Omron CX-Programmer project 新工程 (CX-Programmer 9.73)

# PLC 新PLC1: CPM1(CPM1A) CPU20

## Global symbols (name address type ; comment)
0.00 BOOL  ; 摇动检测
0.01 BOOL  ; 自动
0.02 BOOL  ; 泵手动
0.03 BOOL  ; 摇动手动
0.04 BOOL  ; 超声波手动
0.05 BOOL  ; 阀门手动
0.06 BOOL  ; 循环启动
0.07 BOOL  ; 超声波定时
0.08 BOOL  ; 摇动定时
0.09 BOOL  ; 非常停止
0.10 BOOL  ; 液位检测
0.11 BOOL  ; 过载保护
10.04 BOOL  ; 泵驱动
10.05 BOOL  ; 摇动马达
10.06 BOOL  ; 超声波
10.07 BOOL  ; 卸油阀
15.00 BOOL  ; 液位正常
200.00 BOOL  ; 循环启动了
200.01 BOOL  ; 循环开始指令
200.02 BOOL  ; 泵起动
200.03 BOOL  ; 阀门闭
200.04 BOOL  ; 泵、阀门、液位异常
200.05 BOOL  ; 液有了
200.06 BOOL  ; 液位异常
200.07 BOOL  ; 泵停止
200.09 BOOL  ; 超声波开
200.10 BOOL  ; 超声波关
200.11 BOOL  ; 泵起动2
200.12 BOOL  ; 摇动开
200.13 BOOL  ; 阀门开
200.14 BOOL  ; 泵停止2
201.00 BOOL  ; 喷淋循环启动
201.01 BOOL  ; 喷淋循环开始
201.02 BOOL  ; 阀门闭2
201.03 BOOL  ; 阀门开2
201.04 BOOL  ; 泵起动3
201.05 BOOL  ; 泵停止3
201.07 BOOL  ; 喷淋循环结束
201.08 BOOL  ; 停止位到
201.09 BOOL  ; 摇动异常
201.10 BOOL  ; 液位异常
210.00 BOOL  ; 全异常
5.00 BOOL  ; 转自动
5.01 BOOL  ; 转手动
5.02 BOOL  ; 泵手动开
5.03 BOOL  ; 泵手动关
5.04 BOOL  ; 摇动手动开
5.05 BOOL  ; 摇动手动关
5.06 BOOL  ; 超声波手动开
5.07 BOOL  ; 超声波手动关
5.08 BOOL  ; 阀门手动开
5.09 BOOL  ; 阀门手动关
5.10 BOOL  ; 循环启动指令
DM1000 CHANNEL  ; 摇动计数
TIM017 BOOL  ; 喷淋时间
TIM021 BOOL  ; 全停止

## Program 大摇动 (no task)
; 【项目概况】 / 代码控制超声波清洗机，通过泵驱动、摇动马达、超声波和卸油阀的协同工作，实现工件的清洁。系统支持自动模式和手动模式。 / 系统包括PLC控制器CPM1 CPU20、泵驱动、摇动马达、超声波发生器、卸油阀、液位传感器、过载保护开关和非常停止按钮等物理设备。 / 【运行解析】 / 1.操作员可以通过自动模式选择切换运行模式。 / 2.在自动模式下，按下循环启动按钮会置位清洗循环启动标志。 / 3.在启动清洗循环前，液位传感器必须检测到液位正常标志为真，确保清洗液充足，否则无法启动。 / 4.清洗开始后，泵启动标志激活泵驱动循环清洗液，同时阀门关闭标志关闭卸油阀，保持液位稳定。 / 5.随后，系统进入超声波和摇动阶段，超声波启动标志启动超声波发生器，运行时间由超声波定时开关控制；接着摇动启动标志启动摇动马达，运行时间由摇动定时开关决定。 / 6.系统通过互锁逻辑确保超声波发生器和摇动马达不会同时运行，以避免干扰或设备过载。 / 7.摇动马达运行时，摇动计数器记录频率，若未在规定时间内达到5次，摇动异常标志会置位，表示检测到异常。 / 8.超声波和摇动完成后，喷淋循环启动标志触发喷淋清洗，泵启动3标志再次启动泵驱动，阀门关闭2标志和阀门开启2标志协作控制卸油阀，喷淋时间定时器计时300个单位后，喷淋循环结束标志置位。 / 9.最终，全停止定时器计时结束，停止位到标志置位，所有动作停止。 / 10.在手动模式下，操作员可通过泵手动开关、摇动手动开关、超声波手动开关和阀门手动开关独立控制设备。 / 11.系统通过互锁逻辑确保泵驱动和卸油阀不会同时运行，以防止清洗液同时循环和排放。 / 12.当泵手动开指令和阀门手动开指令同时置位时，系统通过优先级逻辑或互锁机制确保泵驱动和卸油阀不会同时运行。 / 13.系统通过过载保护开关和非常停止按钮监控安全状态，若触发全异常标志，所有动作立即停止。 / 14.同时，清洗循环启动标志和喷淋循环启动标志会复位到初始状态，确保设备安全复位。 / 15.液位异常标志、泵阀液位异常标志或摇动异常标志也能触发全异常标志，提供多重保护。

### Section 段1

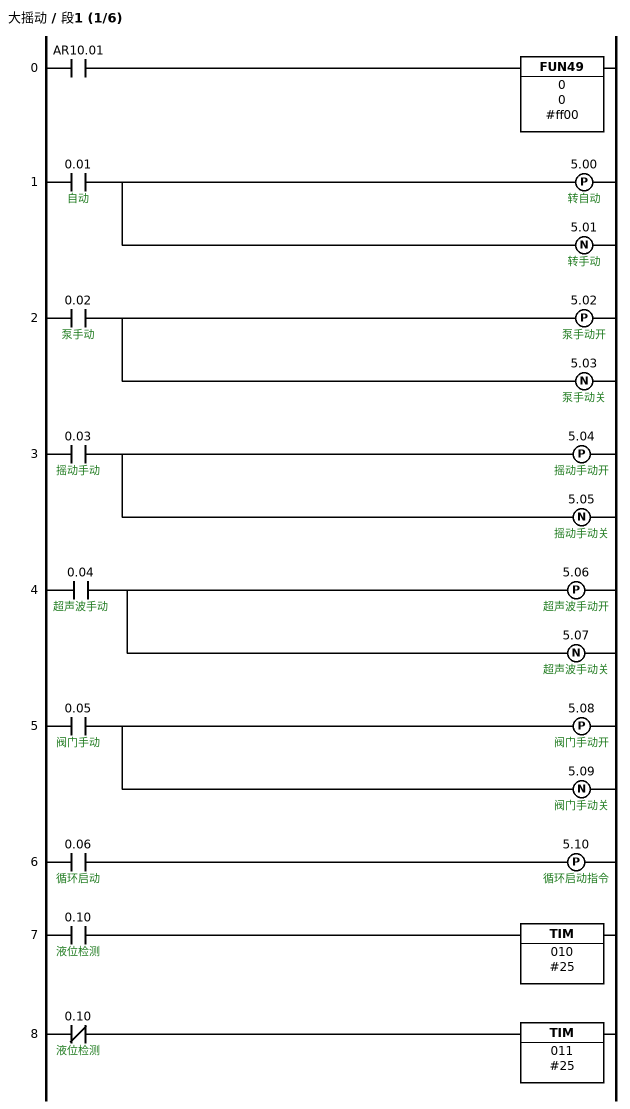
; rung 0
LD AR10.01
FUN49 0 0 #ff00
; rung 1
LD 0.01  ; 自动
DIFU(13) 5.00  ; 转自动
DIFD(14) 5.01  ; 转手动
; rung 2
LD 0.02  ; 泵手动
DIFU(13) 5.02  ; 泵手动开
DIFD(14) 5.03  ; 泵手动关
; rung 3
LD 0.03  ; 摇动手动
DIFU(13) 5.04  ; 摇动手动开
DIFD(14) 5.05  ; 摇动手动关
; rung 4
LD 0.04  ; 超声波手动
DIFU(13) 5.06  ; 超声波手动开
DIFD(14) 5.07  ; 超声波手动关
; rung 5
LD 0.05  ; 阀门手动
DIFU(13) 5.08  ; 阀门手动开
DIFD(14) 5.09  ; 阀门手动关
; rung 6
LD 0.06  ; 循环启动
DIFU(13) 5.10  ; 循环启动指令
; rung 7
LD 0.10  ; 液位检测
TIM 010 #25
; rung 8
LDNOT 0.10  ; 液位检测
TIM 011 #25

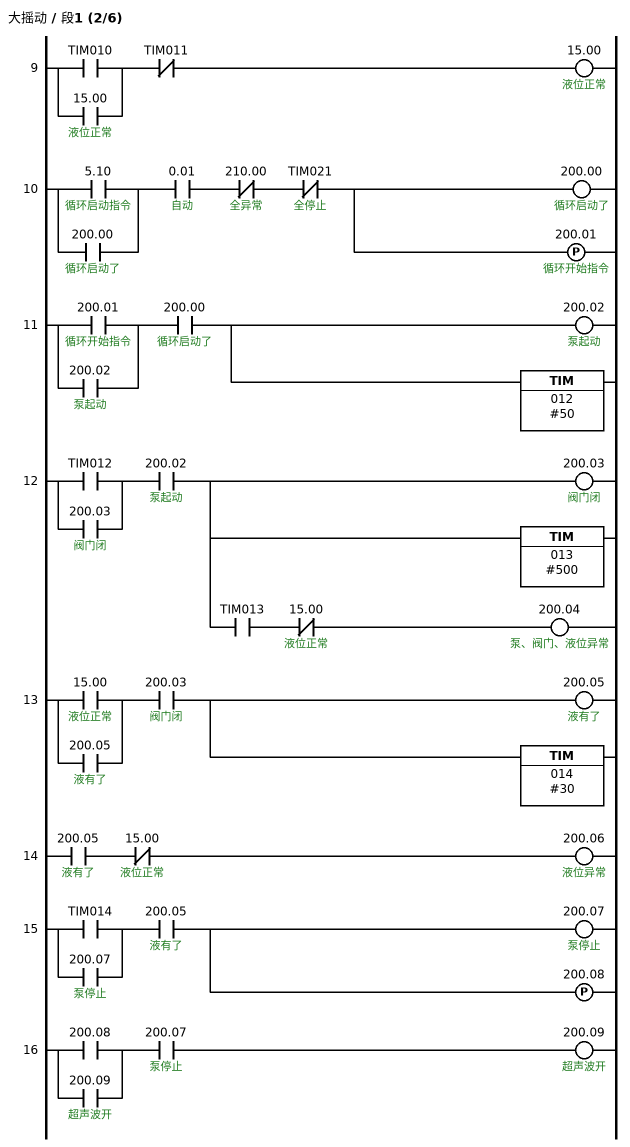
; rung 9
LD TIM010
OR 15.00  ; 液位正常
ANDNOT TIM011
OUT 15.00  ; 液位正常
; rung 10
LD 5.10  ; 循环启动指令
OR 200.00  ; 循环启动了
AND 0.01  ; 自动
ANDNOT 210.00  ; 全异常
ANDNOT TIM021  ; 全停止
OUT 200.00  ; 循环启动了
DIFU(13) 200.01  ; 循环开始指令
; rung 11
LD 200.01  ; 循环开始指令
OR 200.02  ; 泵起动
AND 200.00  ; 循环启动了
OUT 200.02  ; 泵起动
TIM 012 #50
; rung 12
LD TIM012
OR 200.03  ; 阀门闭
AND 200.02  ; 泵起动
OUT 200.03  ; 阀门闭
TIM 013 #500
AND TIM013
ANDNOT 15.00  ; 液位正常
OUT 200.04  ; 泵、阀门、液位异常
; rung 13
LD 15.00  ; 液位正常
OR 200.05  ; 液有了
AND 200.03  ; 阀门闭
OUT 200.05  ; 液有了
TIM 014 #30
; rung 14
LD 200.05  ; 液有了
ANDNOT 15.00  ; 液位正常
OUT 200.06  ; 液位异常
; rung 15
LD TIM014
OR 200.07  ; 泵停止
AND 200.05  ; 液有了
OUT 200.07  ; 泵停止
DIFU(13) 200.08
; rung 16
LD 200.08
OR 200.09  ; 超声波开
AND 200.07  ; 泵停止
OUT 200.09  ; 超声波开

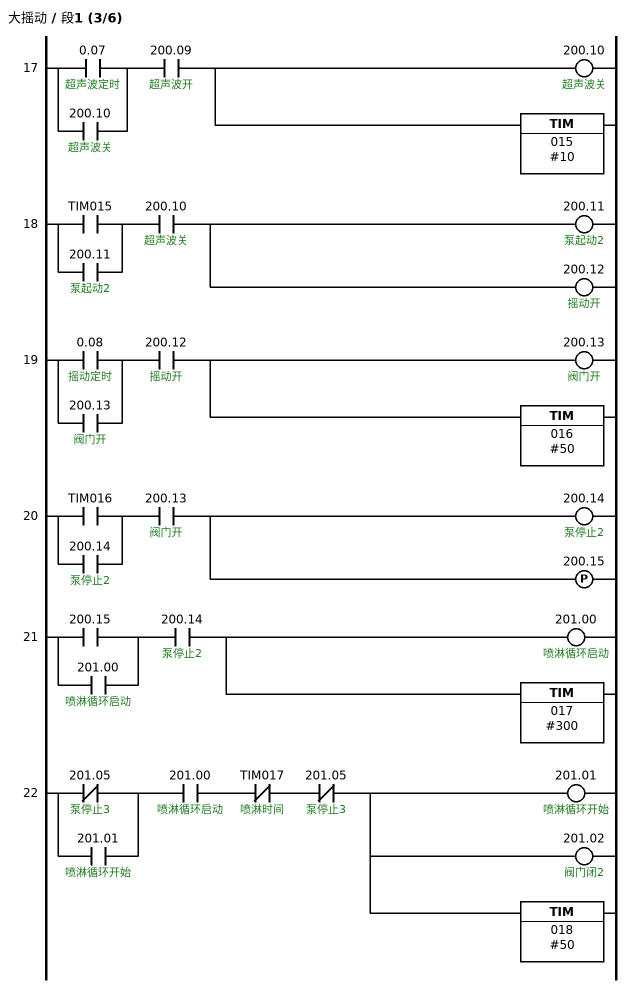
; rung 17
LD 0.07  ; 超声波定时
OR 200.10  ; 超声波关
AND 200.09  ; 超声波开
OUT 200.10  ; 超声波关
TIM 015 #10
; rung 18
LD TIM015
OR 200.11  ; 泵起动2
AND 200.10  ; 超声波关
OUT 200.11  ; 泵起动2
OUT 200.12  ; 摇动开
; rung 19
LD 0.08  ; 摇动定时
OR 200.13  ; 阀门开
AND 200.12  ; 摇动开
OUT 200.13  ; 阀门开
TIM 016 #50
; rung 20
LD TIM016
OR 200.14  ; 泵停止2
AND 200.13  ; 阀门开
OUT 200.14  ; 泵停止2
DIFU(13) 200.15
; rung 21
LD 200.15
OR 201.00  ; 喷淋循环启动
AND 200.14  ; 泵停止2
OUT 201.00  ; 喷淋循环启动
TIM 017 #300
; rung 22
LDNOT 201.05  ; 泵停止3
OR 201.01  ; 喷淋循环开始
AND 201.00  ; 喷淋循环启动
ANDNOT TIM017  ; 喷淋时间
ANDNOT 201.05  ; 泵停止3
OUT 201.01  ; 喷淋循环开始
OUT 201.02  ; 阀门闭2
TIM 018 #50

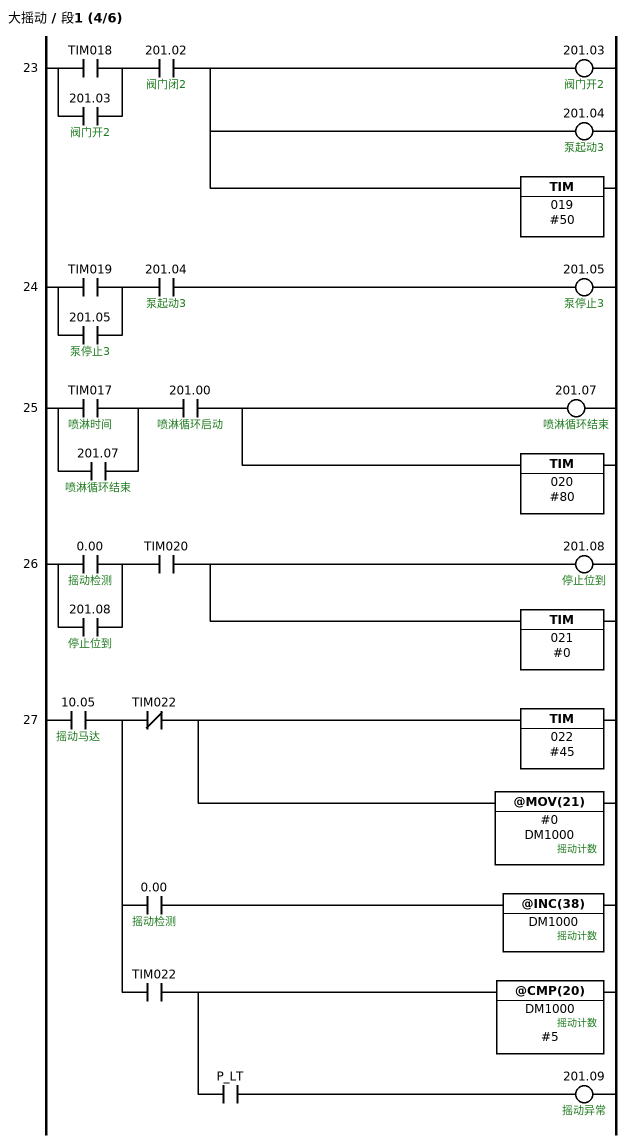
; rung 23
LD TIM018
OR 201.03  ; 阀门开2
AND 201.02  ; 阀门闭2
OUT 201.03  ; 阀门开2
OUT 201.04  ; 泵起动3
TIM 019 #50
; rung 24
LD TIM019
OR 201.05  ; 泵停止3
AND 201.04  ; 泵起动3
OUT 201.05  ; 泵停止3
; rung 25
LD TIM017  ; 喷淋时间
OR 201.07  ; 喷淋循环结束
AND 201.00  ; 喷淋循环启动
OUT 201.07  ; 喷淋循环结束
TIM 020 #80
; rung 26
LD 0.00  ; 摇动检测
OR 201.08  ; 停止位到
AND TIM020
OUT 201.08  ; 停止位到
TIM 021 #0
; rung 27
LD 10.05  ; 摇动马达
OUT TR0
ANDNOT TIM022
TIM 022 #45
@MOV(21) #0 DM1000  ; 摇动计数
LD TR0
AND 0.00  ; 摇动检测
@INC(38) DM1000  ; 摇动计数
LD TR0
AND TIM022
@CMP(20) DM1000 #5  ; 摇动计数
AND P_LT
OUT 201.09  ; 摇动异常

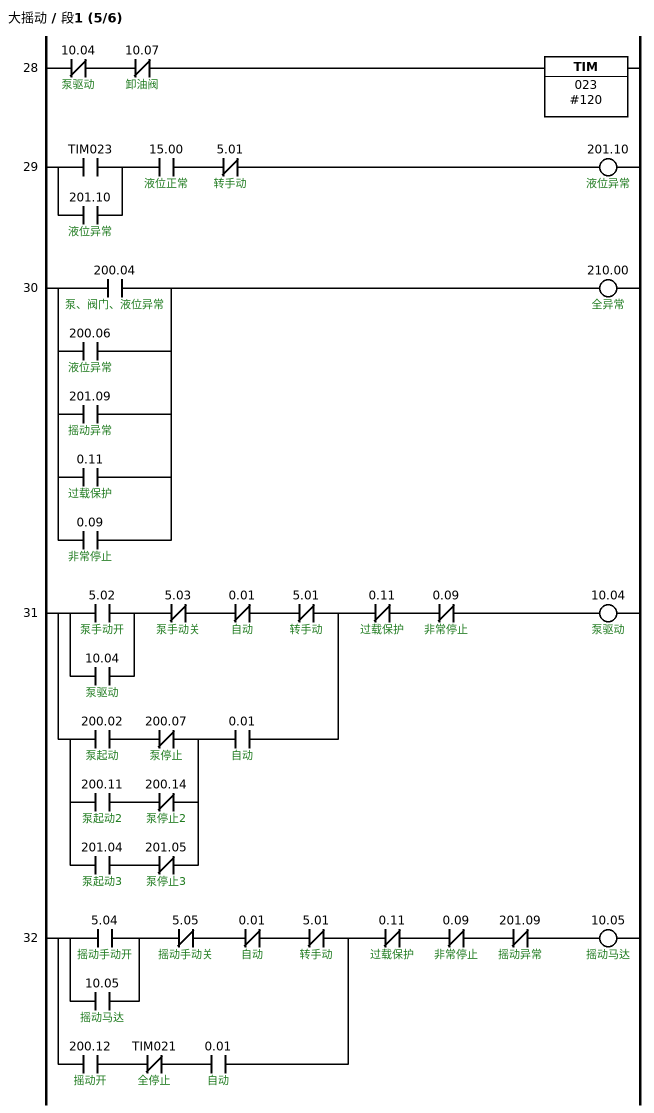
; rung 28
LDNOT 10.04  ; 泵驱动
ANDNOT 10.07  ; 卸油阀
TIM 023 #120
; rung 29
LD TIM023
OR 201.10  ; 液位异常
AND 15.00  ; 液位正常
ANDNOT 5.01  ; 转手动
OUT 201.10  ; 液位异常
; rung 30
LD 200.04  ; 泵、阀门、液位异常
OR 200.06  ; 液位异常
OR 201.09  ; 摇动异常
OR 0.11  ; 过载保护
OR 0.09  ; 非常停止
OUT 210.00  ; 全异常
; rung 31
LD 5.02  ; 泵手动开
OR 10.04  ; 泵驱动
ANDNOT 5.03  ; 泵手动关
ANDNOT 0.01  ; 自动
ANDNOT 5.01  ; 转手动
LD 200.02  ; 泵起动
ANDNOT 200.07  ; 泵停止
LD 200.11  ; 泵起动2
ANDNOT 200.14  ; 泵停止2
ORLD
LD 201.04  ; 泵起动3
ANDNOT 201.05  ; 泵停止3
ORLD
AND 0.01  ; 自动
ORLD
ANDNOT 0.11  ; 过载保护
ANDNOT 0.09  ; 非常停止
OUT 10.04  ; 泵驱动
; rung 32
LD 5.04  ; 摇动手动开
OR 10.05  ; 摇动马达
ANDNOT 5.05  ; 摇动手动关
ANDNOT 0.01  ; 自动
ANDNOT 5.01  ; 转手动
LD 200.12  ; 摇动开
ANDNOT TIM021  ; 全停止
AND 0.01  ; 自动
ORLD
ANDNOT 0.11  ; 过载保护
ANDNOT 0.09  ; 非常停止
ANDNOT 201.09  ; 摇动异常
OUT 10.05  ; 摇动马达

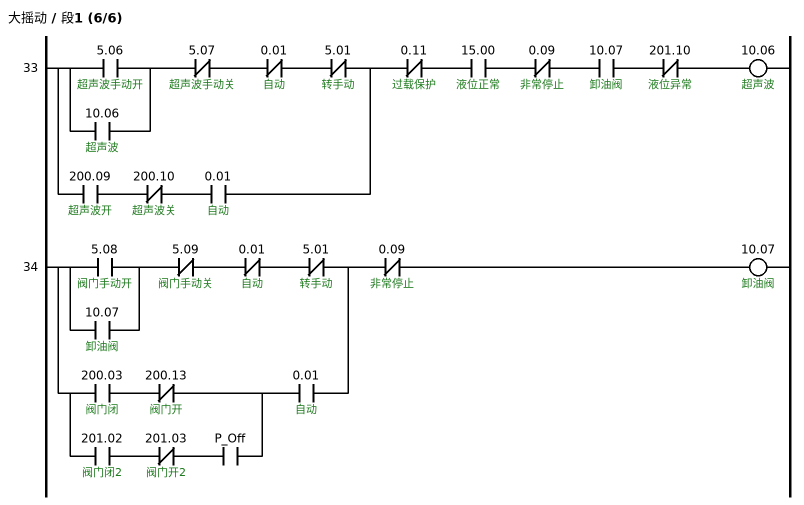
; rung 33
LD 5.06  ; 超声波手动开
OR 10.06  ; 超声波
ANDNOT 5.07  ; 超声波手动关
ANDNOT 0.01  ; 自动
ANDNOT 5.01  ; 转手动
LD 200.09  ; 超声波开
ANDNOT 200.10  ; 超声波关
AND 0.01  ; 自动
ORLD
ANDNOT 0.11  ; 过载保护
AND 15.00  ; 液位正常
ANDNOT 0.09  ; 非常停止
AND 10.07  ; 卸油阀
ANDNOT 201.10  ; 液位异常
OUT 10.06  ; 超声波
; rung 34
LD 5.08  ; 阀门手动开
OR 10.07  ; 卸油阀
ANDNOT 5.09  ; 阀门手动关
ANDNOT 0.01  ; 自动
ANDNOT 5.01  ; 转手动
LD 200.03  ; 阀门闭
ANDNOT 200.13  ; 阀门开
LD 201.02  ; 阀门闭2
ANDNOT 201.03  ; 阀门开2
AND P_Off
ORLD
AND 0.01  ; 自动
ORLD
ANDNOT 0.09  ; 非常停止
OUT 10.07  ; 卸油阀

### Section END
; rung 0
END(01)